# EPICS autosave request: SPApp/Db/VindumController_settings.req
$(P)PumpMode
$(P)TotalVolumeSP
